(* Logix 5000 project; controller Safety vendor 1 type 14 code 148 rev 32.11; software revision 32.03; part 15 of 17 *)
(* tags used below, declared in another part *)
   A1_S20_ModFlt : ALIAS FOR Flt_Modules[0].0;   // A1 Point I/O Slot20 Module Fault (1 = Fault)
   A1_S21_ModFlt : ALIAS FOR Flt_Modules[0].1;   // A1 Point I/O Slot21 Module Fault (1 = Fault)
   C1_S12_ModFlt : ALIAS FOR Flt_Modules[0].2;   // C1 Point I/O Slot12 Module Fault (1 = Fault)
   CHPLC_S1_ModFlt : ALIAS FOR Flt_Modules[0].3;   // CHPLC Point I/O Slot01 Module Fault (1 = Fault)
   CHPLC_S2_ModFlt : ALIAS FOR Flt_Modules[0].4;   // CHPLC Point I/O Slot02 Module Fault (1 = Fault)
   CHPLC_S3_ModFlt : ALIAS FOR Flt_Modules[0].5;   // CHPLC Point I/O Slot03 Module Fault (1 = Fault)
   CHPLC_S4_ModFlt : ALIAS FOR Flt_Modules[0].6;   // CHPLC Point I/O Slot04 Module Fault (1 = Fault)
   CHPLC_S5_ModFlt : ALIAS FOR Flt_Modules[0].7;   // CHPLC Point I/O Slot05 Module Fault (1 = Fault)
   CHPLC_S6_ModFlt : ALIAS FOR Flt_Modules[0].8;   // CHPLC Point I/O Slot06 Module Fault (1 = Fault)
   D1_S12_ModFlt : ALIAS FOR Flt_Modules[0].9;   // D1 Point I/O Slot12 Module Fault (1 = Fault)
   DPD_S14_ModFlt : ALIAS FOR Flt_Modules[0].10;   // DPD Point I/O Slot14 Module Fault (1 = Fault)
   DPD_S15_ModFlt : ALIAS FOR Flt_Modules[0].11;   // DPD Point I/O Slot15 Module Fault (1 = Fault)
   E1_S10_ModFlt : ALIAS FOR Flt_Modules[0].12;   // E1 Point I/O Slot10 Module Fault (1 = Fault)
   F1_S19_ModFlt : ALIAS FOR Flt_Modules[0].13;   // F1 Point I/O Slot19 Module Fault (1 = Fault)
   F1_S20_ModFlt : ALIAS FOR Flt_Modules[0].14;   // F1 Point I/O Slot20 Module Fault (1 = Fault)
   G1_S11_ModFlt : ALIAS FOR Flt_Modules[0].15;   // G1 Point I/O Slot11 Module Fault (1 = Fault)
   G1_S12_ModFlt : ALIAS FOR Flt_Modules[0].16;   // G1 Point I/O Slot12 Module Fault (1 = Fault)
   H1_S5_ModFlt : ALIAS FOR Flt_Modules[0].17;   // H1 Point I/O Slot05 Module Fault (1 = Fault)
   H1_S6_ModFlt : ALIAS FOR Flt_Modules[0].18;   // H1 Point I/O Slot06 Module Fault (1 = Fault)
   Line_TotalMode : BOOL;   // Line TOTAL Mode ( 1= Total Mode) (0 = Coil to Coil)
   LineSts : UDT_SysStatus;
   MCC1_S1_ModFlt : ALIAS FOR Flt_Modules[2].0;   // MCC1 Point I/O Slot01 Module Fault (1 = Fault)
   MCC1_S6_ModFlt : ALIAS FOR Flt_Modules[2].1;   // MCC1 Point I/O Slot06 Module Fault (1 = Fault)
   MCC2_S1_ModFlt : ALIAS FOR Flt_Modules[2].2;   // MCC2 Point I/O Slot01 Module Fault (1 = Fault)
   MCC2_S2_ModFlt : ALIAS FOR Flt_Modules[2].3;   // MCC2 Point I/O Slot02 Module Fault (1 = Fault)
   MCC3_S1_ModFlt : ALIAS FOR Flt_Modules[2].4;   // MCC3 Point I/O Slot01 Module Fault (1 = Fault)
   MCC3_S3_ModFlt : ALIAS FOR Flt_Modules[2].5;   // MCC3 Point I/O Slot03 Module Fault (1 = Fault)
   MCC3_S4_ModFlt : ALIAS FOR Flt_Modules[2].6;   // MCC3 Point I/O Slot04 Module Fault (1 = Fault)
   MCC4_S1_ModFlt : ALIAS FOR Flt_Modules[2].7;   // MCC4 Point I/O Slot01 Module Fault (1 = Fault)
   MCC4_S3_ModFlt : ALIAS FOR Flt_Modules[2].8;   // MCC4 Point I/O Slot03 Module Fault (1 = Fault)
   MCC4_S4_ModFlt : ALIAS FOR Flt_Modules[2].9;   // MCC4 Point I/O Slot04 Module Fault (1 = Fault)
   MCC5_S1_ModFlt : ALIAS FOR Flt_Modules[2].10;   // MCC5 Point I/O Slot01 Module Fault (1 = Fault)
   MCC5_S3_ModFlt : ALIAS FOR Flt_Modules[2].11;   // MCC5 Point I/O Slot03 Module Fault (1 = Fault)
   MCC5_S4_ModFlt : ALIAS FOR Flt_Modules[2].12;   // MCC5 Point I/O Slot04 Module Fault (1 = Fault)
   MCC5_S5_ModFlt : ALIAS FOR Flt_Modules[2].13;   // MCC5 Point I/O Slot05 Module Fault (1 = Fault)
   SDPLC_S1_ModFlt : ALIAS FOR Flt_Modules[0].19;   // SDPLC Point I/O Slot01 Module Fault (1 = Fault)
   SDPLC_S2_ModFlt : ALIAS FOR Flt_Modules[0].20;   // SDPLC Point I/O Slot02 Module Fault (1 = Fault)
   VS2_S10_ModFlt : ALIAS FOR Flt_Modules[0].21;   // VS2 Point I/O Slot10 Module Fault (1 = Fault)
(* System, continued *)

ROUTINE A02_SftyModFlts_GenIO   (* ladder *)
// General I/O
// Safety Module Faults
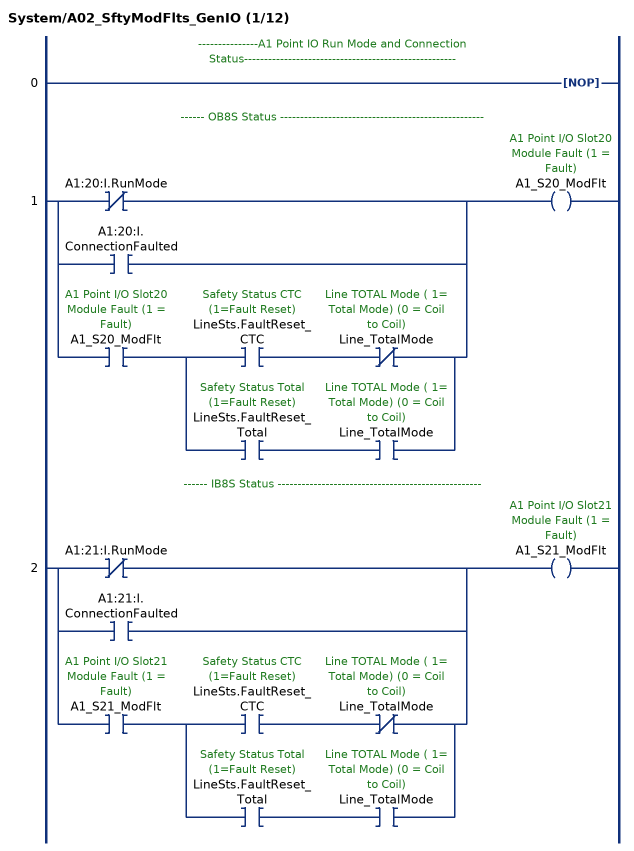
   // ---------------A1 Point IO Run Mode and Connection Status-----------------------------------------------------
   0: NOP();
   // ------ OB8S Status ---------------------------------------------------
   1: [XIO(A1:20:I.RunMode) ,XIC(A1:20:I.ConnectionFaulted) ,XIC(A1_S20_ModFlt) [XIC(LineSts.FaultReset_CTC) XIO(Line_TotalMode) ,XIC(LineSts.FaultReset_Total) XIC(Line_TotalMode) ] ]OTE(A1_S20_ModFlt);
   // ------ IB8S Status ---------------------------------------------------
   2: [XIO(A1:21:I.RunMode) ,XIC(A1:21:I.ConnectionFaulted) ,XIC(A1_S21_ModFlt) [XIC(LineSts.FaultReset_CTC) XIO(Line_TotalMode) ,XIC(LineSts.FaultReset_Total) XIC(Line_TotalMode) ] ]OTE(A1_S21_ModFlt);
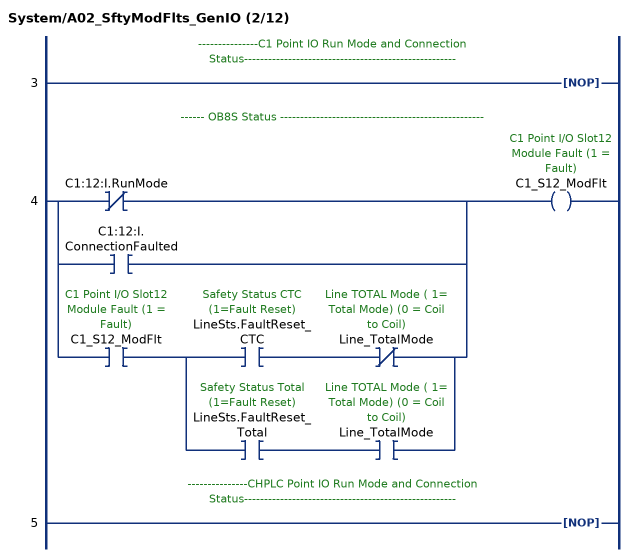
   // ---------------C1 Point IO Run Mode and Connection Status-----------------------------------------------------
   3: NOP();
   // ------ OB8S Status ---------------------------------------------------
   4: [XIO(C1:12:I.RunMode) ,XIC(C1:12:I.ConnectionFaulted) ,XIC(C1_S12_ModFlt) [XIC(LineSts.FaultReset_CTC) XIO(Line_TotalMode) ,XIC(LineSts.FaultReset_Total) XIC(Line_TotalMode) ] ]OTE(C1_S12_ModFlt);
   // ---------------CHPLC Point IO Run Mode and Connection Status-----------------------------------------------------
   5: NOP();
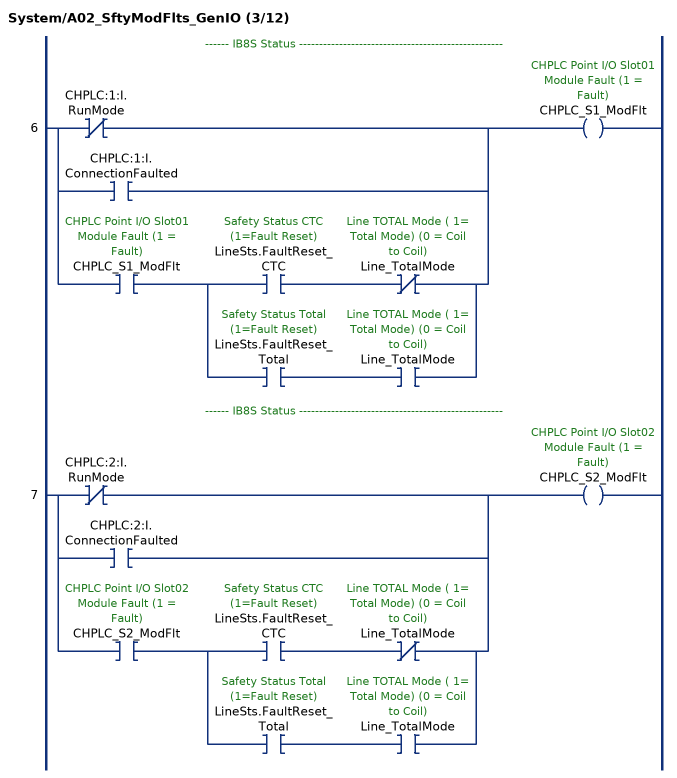
   // ------ IB8S Status ---------------------------------------------------
   6: [XIO(CHPLC:1:I.RunMode) ,XIC(CHPLC:1:I.ConnectionFaulted) ,XIC(CHPLC_S1_ModFlt) [XIC(LineSts.FaultReset_CTC) XIO(Line_TotalMode) ,XIC(LineSts.FaultReset_Total) XIC(Line_TotalMode) ] ]OTE(CHPLC_S1_ModFlt);
   // ------ IB8S Status ---------------------------------------------------
   7: [XIO(CHPLC:2:I.RunMode) ,XIC(CHPLC:2:I.ConnectionFaulted) ,XIC(CHPLC_S2_ModFlt) [XIC(LineSts.FaultReset_CTC) XIO(Line_TotalMode) ,XIC(LineSts.FaultReset_Total) XIC(Line_TotalMode) ] ]OTE(CHPLC_S2_ModFlt);
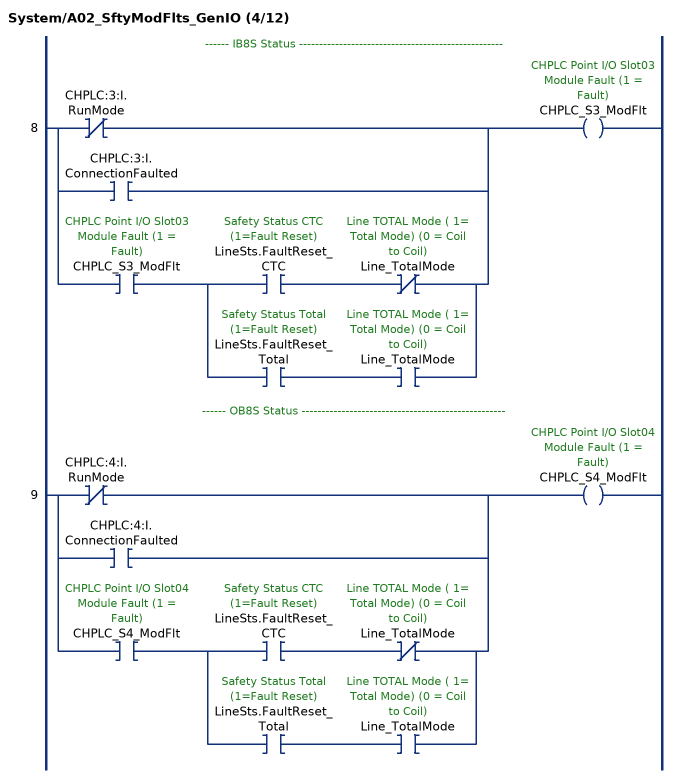
   // ------ IB8S Status ---------------------------------------------------
   8: [XIO(CHPLC:3:I.RunMode) ,XIC(CHPLC:3:I.ConnectionFaulted) ,XIC(CHPLC_S3_ModFlt) [XIC(LineSts.FaultReset_CTC) XIO(Line_TotalMode) ,XIC(LineSts.FaultReset_Total) XIC(Line_TotalMode) ] ]OTE(CHPLC_S3_ModFlt);
   // ------ OB8S Status ---------------------------------------------------
   9: [XIO(CHPLC:4:I.RunMode) ,XIC(CHPLC:4:I.ConnectionFaulted) ,XIC(CHPLC_S4_ModFlt) [XIC(LineSts.FaultReset_CTC) XIO(Line_TotalMode) ,XIC(LineSts.FaultReset_Total) XIC(Line_TotalMode) ] ]OTE(CHPLC_S4_ModFlt);
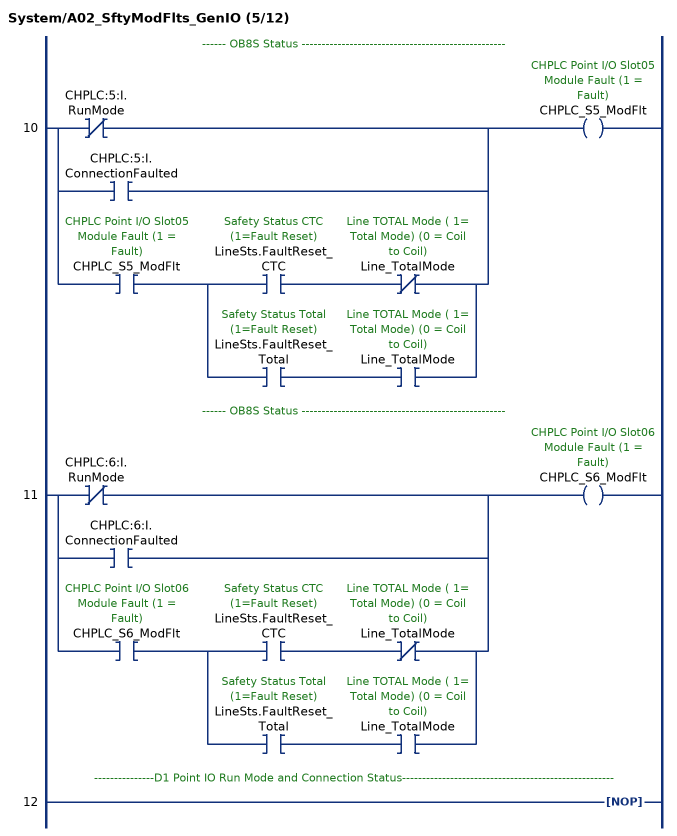
   // ------ OB8S Status ---------------------------------------------------
   10: [XIO(CHPLC:5:I.RunMode) ,XIC(CHPLC:5:I.ConnectionFaulted) ,XIC(CHPLC_S5_ModFlt) [XIC(LineSts.FaultReset_CTC) XIO(Line_TotalMode) ,XIC(LineSts.FaultReset_Total) XIC(Line_TotalMode) ] ]OTE(CHPLC_S5_ModFlt);
   // ------ OB8S Status ---------------------------------------------------
   11: [XIO(CHPLC:6:I.RunMode) ,XIC(CHPLC:6:I.ConnectionFaulted) ,XIC(CHPLC_S6_ModFlt) [XIC(LineSts.FaultReset_CTC) XIO(Line_TotalMode) ,XIC(LineSts.FaultReset_Total) XIC(Line_TotalMode) ] ]OTE(CHPLC_S6_ModFlt);
   // ---------------D1 Point IO Run Mode and Connection Status-----------------------------------------------------
   12: NOP();
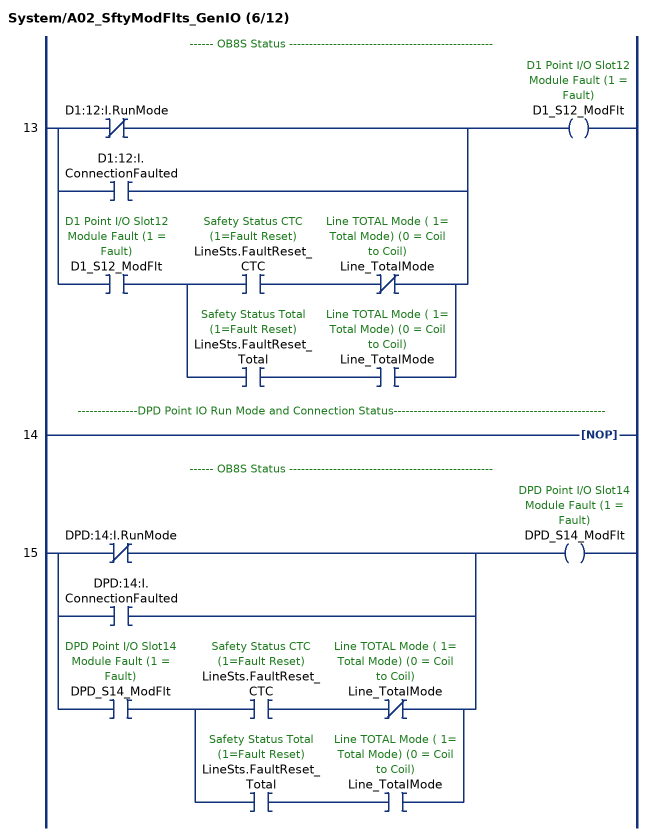
   // ------ OB8S Status ---------------------------------------------------
   13: [XIO(D1:12:I.RunMode) ,XIC(D1:12:I.ConnectionFaulted) ,XIC(D1_S12_ModFlt) [XIC(LineSts.FaultReset_CTC) XIO(Line_TotalMode) ,XIC(LineSts.FaultReset_Total) XIC(Line_TotalMode) ] ]OTE(D1_S12_ModFlt);
   // ---------------DPD Point IO Run Mode and Connection Status-----------------------------------------------------
   14: NOP();
   // ------ OB8S Status ---------------------------------------------------
   15: [XIO(DPD:14:I.RunMode) ,XIC(DPD:14:I.ConnectionFaulted) ,XIC(DPD_S14_ModFlt) [XIC(LineSts.FaultReset_CTC) XIO(Line_TotalMode) ,XIC(LineSts.FaultReset_Total) XIC(Line_TotalMode) ] ]OTE(DPD_S14_ModFlt);
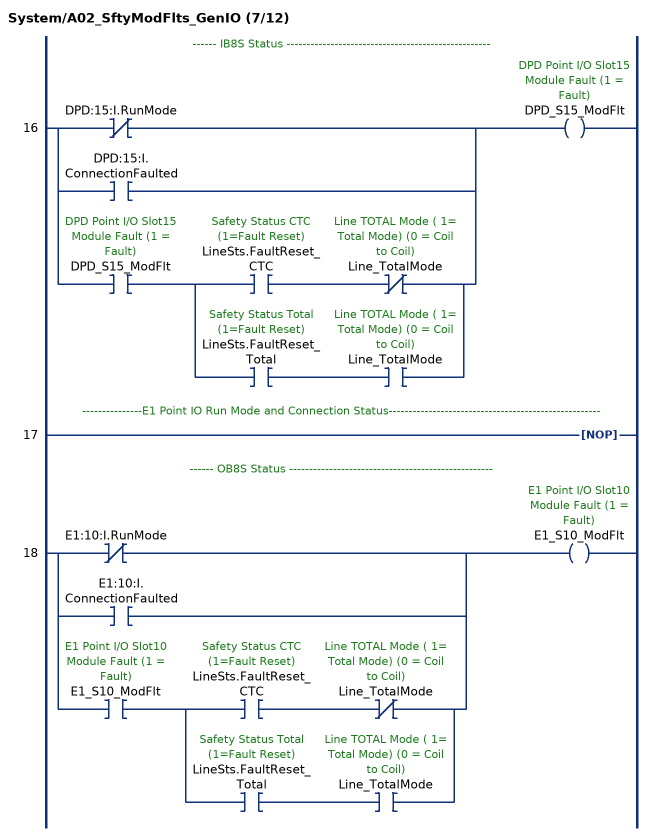
   // ------ IB8S Status ---------------------------------------------------
   16: [XIO(DPD:15:I.RunMode) ,XIC(DPD:15:I.ConnectionFaulted) ,XIC(DPD_S15_ModFlt) [XIC(LineSts.FaultReset_CTC) XIO(Line_TotalMode) ,XIC(LineSts.FaultReset_Total) XIC(Line_TotalMode) ] ]OTE(DPD_S15_ModFlt);
   // ---------------E1 Point IO Run Mode and Connection Status-----------------------------------------------------
   17: NOP();
   // ------ OB8S Status ---------------------------------------------------
   18: [XIO(E1:10:I.RunMode) ,XIC(E1:10:I.ConnectionFaulted) ,XIC(E1_S10_ModFlt) [XIC(LineSts.FaultReset_CTC) XIO(Line_TotalMode) ,XIC(LineSts.FaultReset_Total) XIC(Line_TotalMode) ] ]OTE(E1_S10_ModFlt);
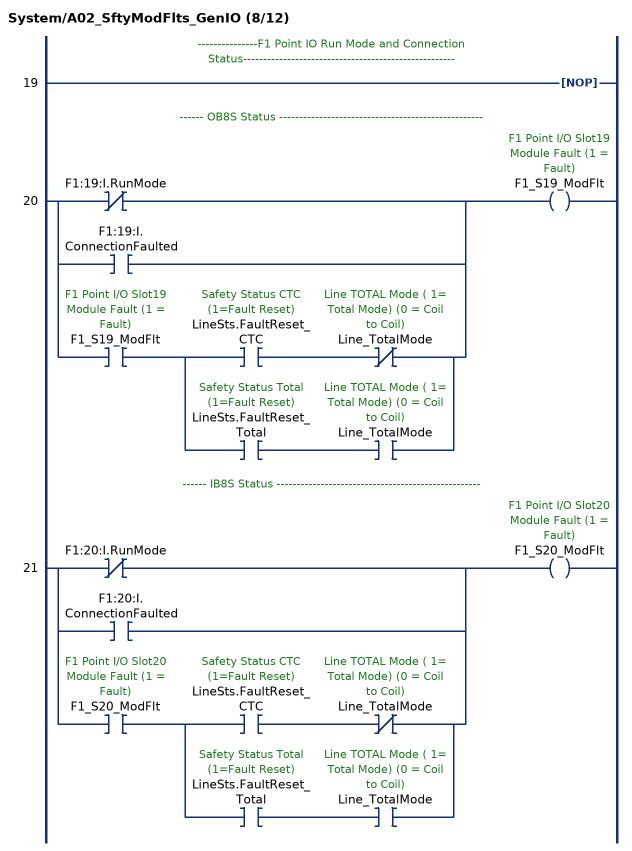
   // ---------------F1 Point IO Run Mode and Connection Status-----------------------------------------------------
   19: NOP();
   // ------ OB8S Status ---------------------------------------------------
   20: [XIO(F1:19:I.RunMode) ,XIC(F1:19:I.ConnectionFaulted) ,XIC(F1_S19_ModFlt) [XIC(LineSts.FaultReset_CTC) XIO(Line_TotalMode) ,XIC(LineSts.FaultReset_Total) XIC(Line_TotalMode) ] ]OTE(F1_S19_ModFlt);
   // ------ IB8S Status ---------------------------------------------------
   21: [XIO(F1:20:I.RunMode) ,XIC(F1:20:I.ConnectionFaulted) ,XIC(F1_S20_ModFlt) [XIC(LineSts.FaultReset_CTC) XIO(Line_TotalMode) ,XIC(LineSts.FaultReset_Total) XIC(Line_TotalMode) ] ]OTE(F1_S20_ModFlt);
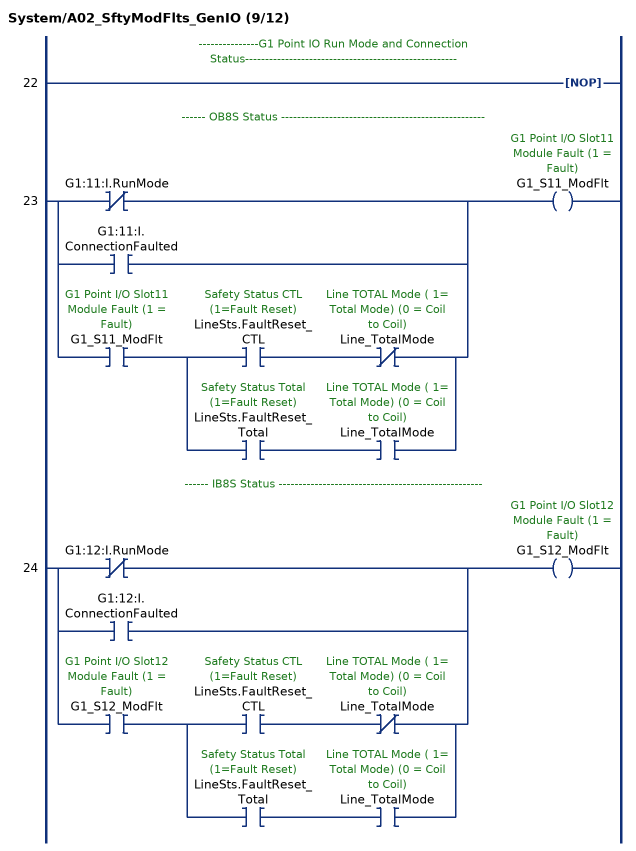
   // ---------------G1 Point IO Run Mode and Connection Status-----------------------------------------------------
   22: NOP();
   // ------ OB8S Status ---------------------------------------------------
   23: [XIO(G1:11:I.RunMode) ,XIC(G1:11:I.ConnectionFaulted) ,XIC(G1_S11_ModFlt) [XIC(LineSts.FaultReset_CTL) XIO(Line_TotalMode) ,XIC(LineSts.FaultReset_Total) XIC(Line_TotalMode) ] ]OTE(G1_S11_ModFlt);
   // ------ IB8S Status ---------------------------------------------------
   24: [XIO(G1:12:I.RunMode) ,XIC(G1:12:I.ConnectionFaulted) ,XIC(G1_S12_ModFlt) [XIC(LineSts.FaultReset_CTL) XIO(Line_TotalMode) ,XIC(LineSts.FaultReset_Total) XIC(Line_TotalMode) ] ]OTE(G1_S12_ModFlt);
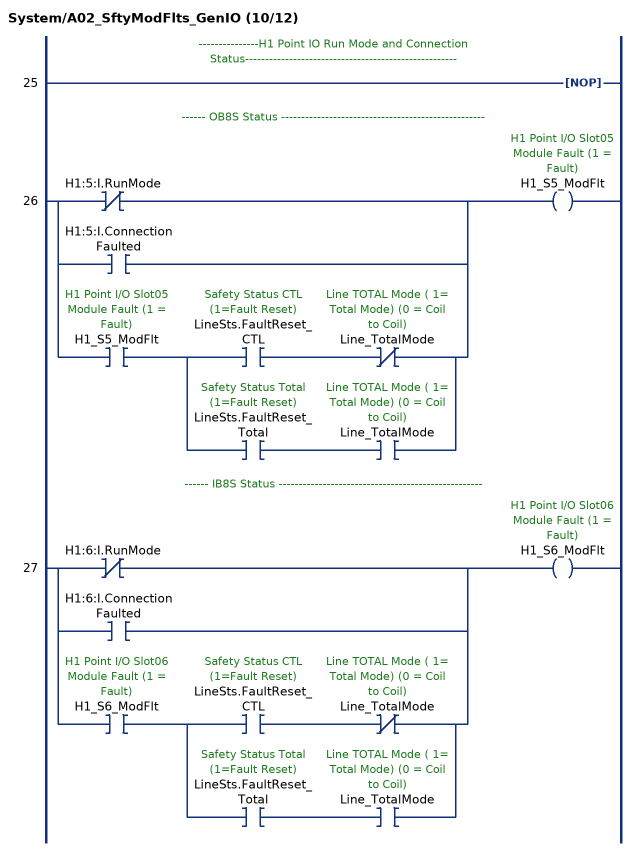
   // ---------------H1 Point IO Run Mode and Connection Status-----------------------------------------------------
   25: NOP();
   // ------ OB8S Status ---------------------------------------------------
   26: [XIO(H1:5:I.RunMode) ,XIC(H1:5:I.ConnectionFaulted) ,XIC(H1_S5_ModFlt) [XIC(LineSts.FaultReset_CTL) XIO(Line_TotalMode) ,XIC(LineSts.FaultReset_Total) XIC(Line_TotalMode) ] ]OTE(H1_S5_ModFlt);
   // ------ IB8S Status ---------------------------------------------------
   27: [XIO(H1:6:I.RunMode) ,XIC(H1:6:I.ConnectionFaulted) ,XIC(H1_S6_ModFlt) [XIC(LineSts.FaultReset_CTL) XIO(Line_TotalMode) ,XIC(LineSts.FaultReset_Total) XIC(Line_TotalMode) ] ]OTE(H1_S6_ModFlt);
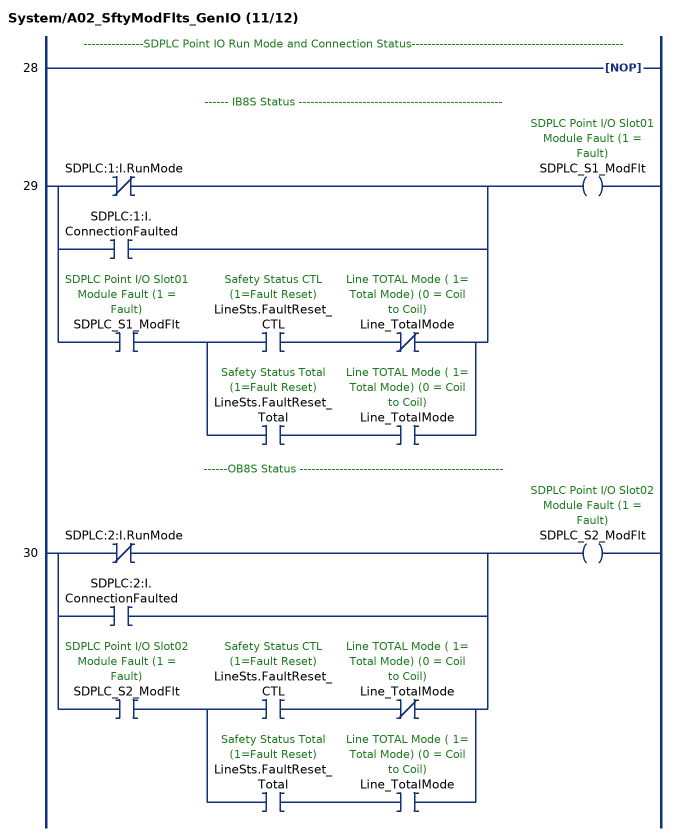
   // ---------------SDPLC Point IO Run Mode and Connection Status-----------------------------------------------------
   28: NOP();
   // ------ IB8S Status ---------------------------------------------------
   29: [XIO(SDPLC:1:I.RunMode) ,XIC(SDPLC:1:I.ConnectionFaulted) ,XIC(SDPLC_S1_ModFlt) [XIC(LineSts.FaultReset_CTL) XIO(Line_TotalMode) ,XIC(LineSts.FaultReset_Total) XIC(Line_TotalMode) ] ]OTE(SDPLC_S1_ModFlt);
   // ------OB8S Status ---------------------------------------------------
   30: [XIO(SDPLC:2:I.RunMode) ,XIC(SDPLC:2:I.ConnectionFaulted) ,XIC(SDPLC_S2_ModFlt) [XIC(LineSts.FaultReset_CTL) XIO(Line_TotalMode) ,XIC(LineSts.FaultReset_Total) XIC(Line_TotalMode) ] ]OTE(SDPLC_S2_ModFlt);
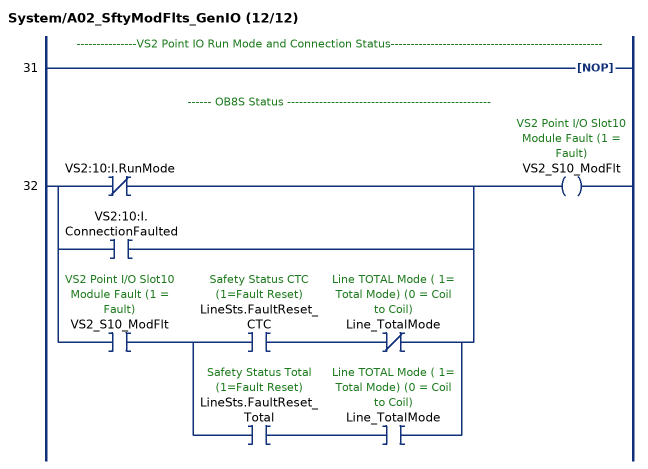
   // ---------------VS2 Point IO Run Mode and Connection Status-----------------------------------------------------
   31: NOP();
   // ------ OB8S Status ---------------------------------------------------
   32: [XIO(VS2:10:I.RunMode) ,XIC(VS2:10:I.ConnectionFaulted) ,XIC(VS2_S10_ModFlt) [XIC(LineSts.FaultReset_CTC) XIO(Line_TotalMode) ,XIC(LineSts.FaultReset_Total) XIC(Line_TotalMode) ] ]OTE(VS2_S10_ModFlt);
END_ROUTINE

ROUTINE A03_SftyModFlts_MCC   (* ladder *)
// MCC
// Safety Module Faults
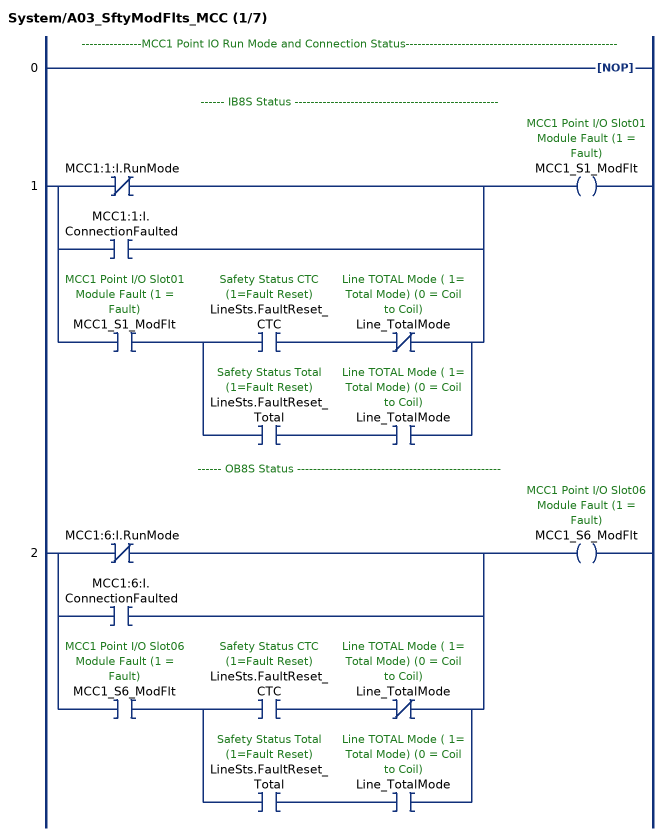
   // ---------------MCC1 Point IO Run Mode and Connection Status-----------------------------------------------------
   0: NOP();
   // ------ IB8S Status ---------------------------------------------------
   1: [XIO(MCC1:1:I.RunMode) ,XIC(MCC1:1:I.ConnectionFaulted) ,XIC(MCC1_S1_ModFlt) [XIC(LineSts.FaultReset_CTC) XIO(Line_TotalMode) ,XIC(LineSts.FaultReset_Total) XIC(Line_TotalMode) ] ]OTE(MCC1_S1_ModFlt);
   // ------ OB8S Status ---------------------------------------------------
   2: [XIO(MCC1:6:I.RunMode) ,XIC(MCC1:6:I.ConnectionFaulted) ,XIC(MCC1_S6_ModFlt) [XIC(LineSts.FaultReset_CTC) XIO(Line_TotalMode) ,XIC(LineSts.FaultReset_Total) XIC(Line_TotalMode) ] ]OTE(MCC1_S6_ModFlt);
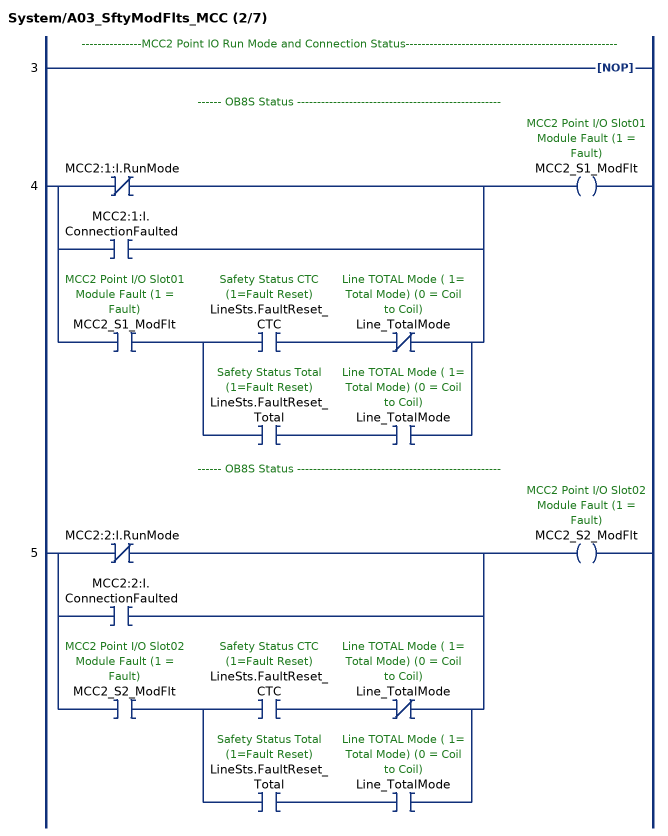
   // ---------------MCC2 Point IO Run Mode and Connection Status-----------------------------------------------------
   3: NOP();
   // ------ OB8S Status ---------------------------------------------------
   4: [XIO(MCC2:1:I.RunMode) ,XIC(MCC2:1:I.ConnectionFaulted) ,XIC(MCC2_S1_ModFlt) [XIC(LineSts.FaultReset_CTC) XIO(Line_TotalMode) ,XIC(LineSts.FaultReset_Total) XIC(Line_TotalMode) ] ]OTE(MCC2_S1_ModFlt);
   // ------ OB8S Status ---------------------------------------------------
   5: [XIO(MCC2:2:I.RunMode) ,XIC(MCC2:2:I.ConnectionFaulted) ,XIC(MCC2_S2_ModFlt) [XIC(LineSts.FaultReset_CTC) XIO(Line_TotalMode) ,XIC(LineSts.FaultReset_Total) XIC(Line_TotalMode) ] ]OTE(MCC2_S2_ModFlt);
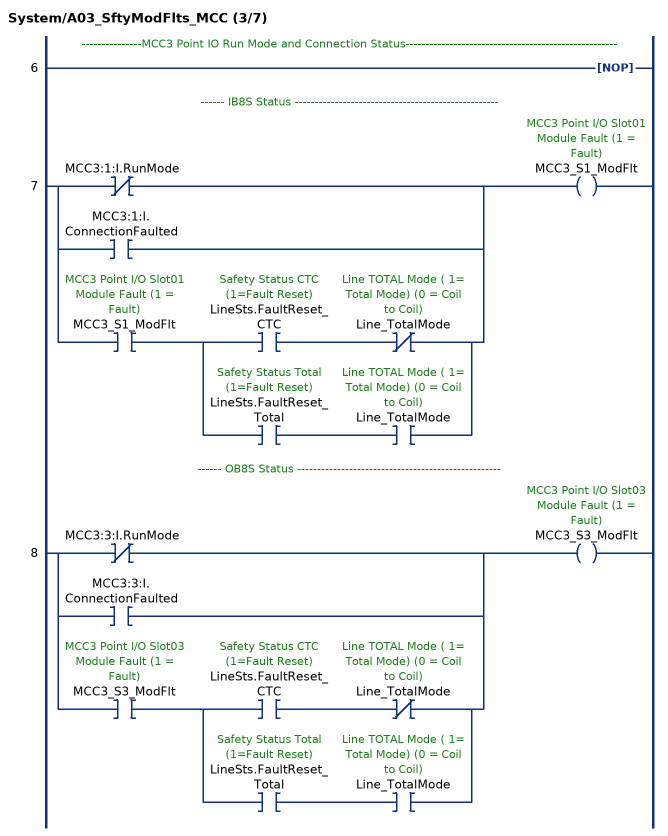
   // ---------------MCC3 Point IO Run Mode and Connection Status-----------------------------------------------------
   6: NOP();
   // ------ IB8S Status ---------------------------------------------------
   7: [XIO(MCC3:1:I.RunMode) ,XIC(MCC3:1:I.ConnectionFaulted) ,XIC(MCC3_S1_ModFlt) [XIC(LineSts.FaultReset_CTC) XIO(Line_TotalMode) ,XIC(LineSts.FaultReset_Total) XIC(Line_TotalMode) ] ]OTE(MCC3_S1_ModFlt);
   // ------ OB8S Status ---------------------------------------------------
   8: [XIO(MCC3:3:I.RunMode) ,XIC(MCC3:3:I.ConnectionFaulted) ,XIC(MCC3_S3_ModFlt) [XIC(LineSts.FaultReset_CTC) XIO(Line_TotalMode) ,XIC(LineSts.FaultReset_Total) XIC(Line_TotalMode) ] ]OTE(MCC3_S3_ModFlt);
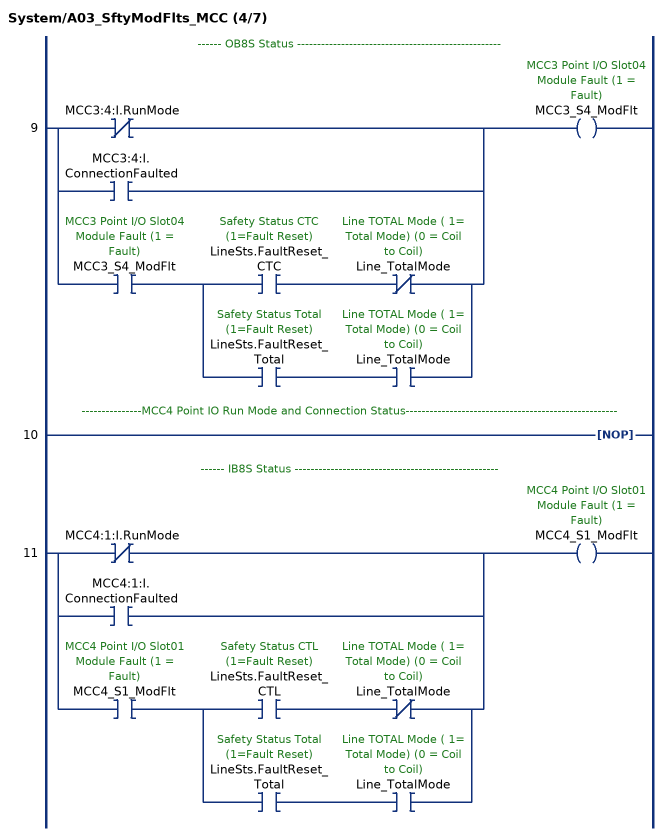
   // ------ OB8S Status ---------------------------------------------------
   9: [XIO(MCC3:4:I.RunMode) ,XIC(MCC3:4:I.ConnectionFaulted) ,XIC(MCC3_S4_ModFlt) [XIC(LineSts.FaultReset_CTC) XIO(Line_TotalMode) ,XIC(LineSts.FaultReset_Total) XIC(Line_TotalMode) ] ]OTE(MCC3_S4_ModFlt);
   // ---------------MCC4 Point IO Run Mode and Connection Status-----------------------------------------------------
   10: NOP();
   // ------ IB8S Status ---------------------------------------------------
   11: [XIO(MCC4:1:I.RunMode) ,XIC(MCC4:1:I.ConnectionFaulted) ,XIC(MCC4_S1_ModFlt) [XIC(LineSts.FaultReset_CTL) XIO(Line_TotalMode) ,XIC(LineSts.FaultReset_Total) XIC(Line_TotalMode) ] ]OTE(MCC4_S1_ModFlt);
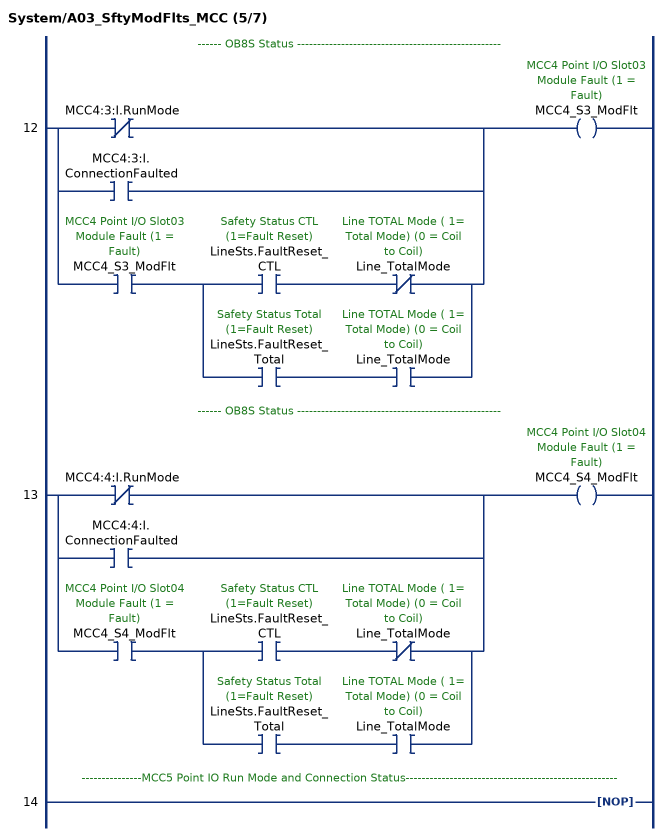
   // ------ OB8S Status ---------------------------------------------------
   12: [XIO(MCC4:3:I.RunMode) ,XIC(MCC4:3:I.ConnectionFaulted) ,XIC(MCC4_S3_ModFlt) [XIC(LineSts.FaultReset_CTL) XIO(Line_TotalMode) ,XIC(LineSts.FaultReset_Total) XIC(Line_TotalMode) ] ]OTE(MCC4_S3_ModFlt);
   // ------ OB8S Status ---------------------------------------------------
   13: [XIO(MCC4:4:I.RunMode) ,XIC(MCC4:4:I.ConnectionFaulted) ,XIC(MCC4_S4_ModFlt) [XIC(LineSts.FaultReset_CTL) XIO(Line_TotalMode) ,XIC(LineSts.FaultReset_Total) XIC(Line_TotalMode) ] ]OTE(MCC4_S4_ModFlt);
   // ---------------MCC5 Point IO Run Mode and Connection Status-----------------------------------------------------
   14: NOP();
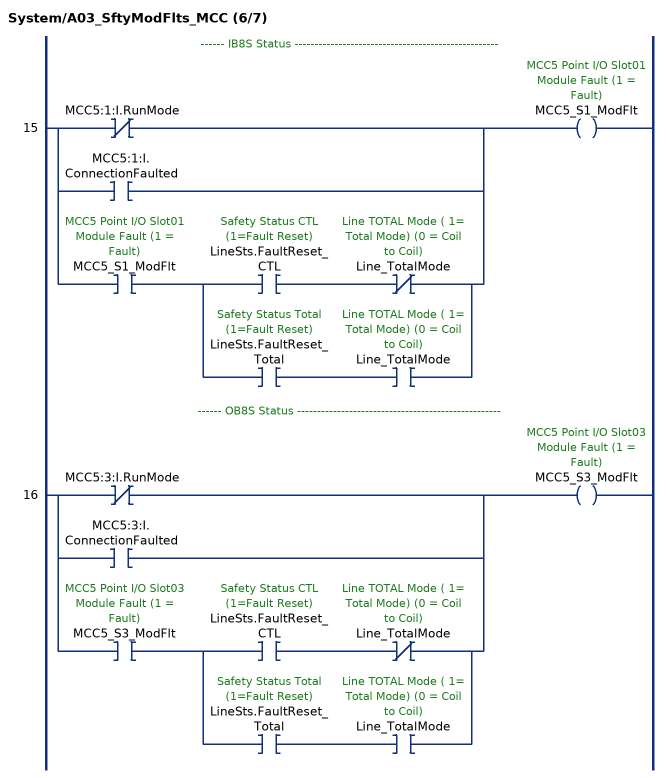
   // ------ IB8S Status ---------------------------------------------------
   15: [XIO(MCC5:1:I.RunMode) ,XIC(MCC5:1:I.ConnectionFaulted) ,XIC(MCC5_S1_ModFlt) [XIC(LineSts.FaultReset_CTL) XIO(Line_TotalMode) ,XIC(LineSts.FaultReset_Total) XIC(Line_TotalMode) ] ]OTE(MCC5_S1_ModFlt);
   // ------ OB8S Status ---------------------------------------------------
   16: [XIO(MCC5:3:I.RunMode) ,XIC(MCC5:3:I.ConnectionFaulted) ,XIC(MCC5_S3_ModFlt) [XIC(LineSts.FaultReset_CTL) XIO(Line_TotalMode) ,XIC(LineSts.FaultReset_Total) XIC(Line_TotalMode) ] ]OTE(MCC5_S3_ModFlt);
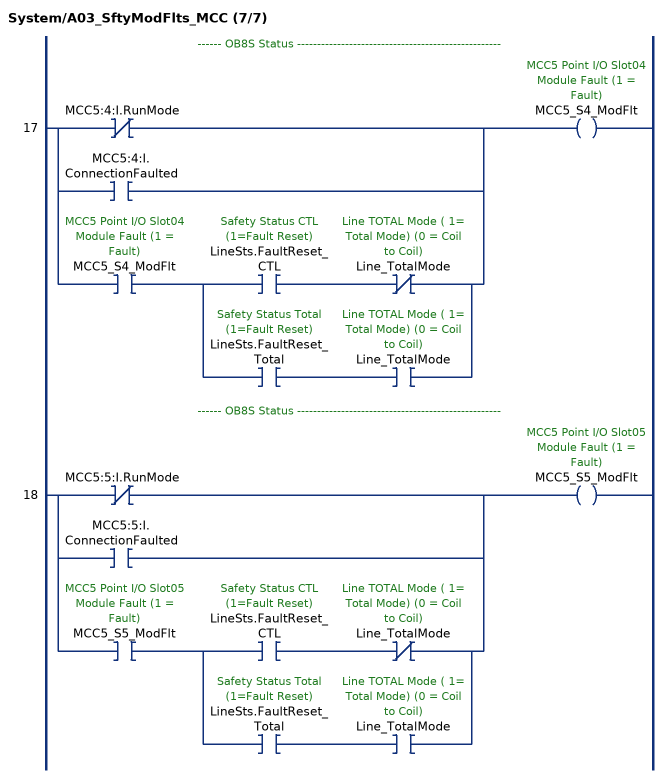
   // ------ OB8S Status ---------------------------------------------------
   17: [XIO(MCC5:4:I.RunMode) ,XIC(MCC5:4:I.ConnectionFaulted) ,XIC(MCC5_S4_ModFlt) [XIC(LineSts.FaultReset_CTL) XIO(Line_TotalMode) ,XIC(LineSts.FaultReset_Total) XIC(Line_TotalMode) ] ]OTE(MCC5_S4_ModFlt);
   // ------ OB8S Status ---------------------------------------------------
   18: [XIO(MCC5:5:I.RunMode) ,XIC(MCC5:5:I.ConnectionFaulted) ,XIC(MCC5_S5_ModFlt) [XIC(LineSts.FaultReset_CTL) XIO(Line_TotalMode) ,XIC(LineSts.FaultReset_Total) XIC(Line_TotalMode) ] ]OTE(MCC5_S5_ModFlt);
END_ROUTINE
